// TIA Portal V16 export
// export: Created 2024-05-10T06:46:40.936398Z, ExportSetting WithDefaults, DisplayName Totally Integrated Automation Portal, DisplayVersion V16, DisplayName TIA Portal Version Control Interface, DisplayVersion V16, DisplayName TIA Portal Openness, DisplayVersion V16, DisplayName STEP 7 Professional, DisplayVersion V16, DisplayName STEP 7 Safety, DisplayVersion V16, DisplayName WinCC Professional, DisplayVersion V16
FUNCTION_BLOCK "K05_模式"   // FB5, LAD
{ S7_Optimized_Access := 'TRUE' }
VERSION : 0.1
// stored: AutoNumber false, IsIECCheckEnabled false, IsRetainMemResEnabled false, MemoryReserve 100, SetENOAutomatically false, UDAEnableTagReadback false
   VAR_TEMP   // added for the SCL form of the ladder/FBD networks
      _w1 : Bool;
      _w2 : Bool;
   END_VAR
BEGIN

REGION Network 1: 手动自动模式切换
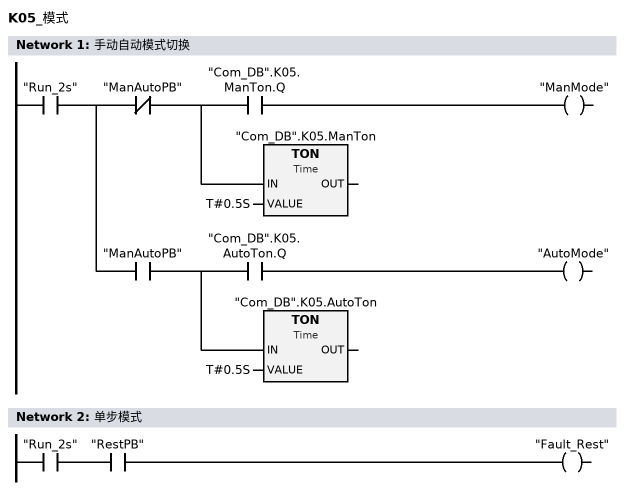
   #_w1 := "Run_2s" AND NOT "ManAutoPB";
   "ManMode" := #_w1 AND "Com_DB".K05.ManTon.Q;
   "Com_DB".K05.ManTon.TON(IN := #_w1, PT := T#0.5S);   // TON coil
   #_w2 := "Run_2s" AND "ManAutoPB";
   "AutoMode" := #_w2 AND "Com_DB".K05.AutoTon.Q;
   "Com_DB".K05.AutoTon.TON(IN := #_w2, PT := T#0.5S);   // TON coil
END_REGION

REGION Network 2: 单步模式
   RUNG wire#powerrail
      Contact( "Run_2s" )
      Contact( "RestPB" )
      Coil( "Fault_Rest" )
   END_RUNG
   // the same network as SCL:
   "Fault_Rest" := "Run_2s" AND "RestPB";
END_REGION

REGION Network 3: 耐久模式
END_REGION
END_FUNCTION_BLOCK
